{attribute 'qualified_only'}
VAR_GLOBAL CONSTANT
	nMaximumSizeOfArray : INT := 20;
END_VAR

(* stored: Version 1.1.0.1, ProductVersion 3.1.4024.16
   GVL GVL: Id {1e2d1b9a-808c-4799-86fc-061f146a77b1} *)
